{attribute 'linkalways'} 
{attribute 'no_explicit_call' := 'This FB is a CLASS and must be accessed using methods or properties'}
{attribute 'enable_dynamic_creation'}
FUNCTION_BLOCK GetBlueprintsVisitor IMPLEMENTS I_NodeFactoryVisitor, I_NodePrototypeVisitor, I_NodeVisitor, I_ExtensionVisitor, I_InputPortVisitor, I_OutputPortVisitor, I_MetadataVisitor, I_ContentVisitor, I_ParameterVisitor, I_AlarmVisitor
VAR
	serializer : I_Serializer;
END_VAR

METHOD PUBLIC Initialize
VAR_INPUT
	Serializer : I_Serializer;
END_VAR
THIS^.serializer := Serializer;
END_METHOD

METHOD VisitAlarm
VAR_INPUT
	VisitingAlarm : I_Alarm;
END_VAR
serializer.AddString(VisitingAlarm.Message);
END_METHOD

METHOD VisitContent
VAR_INPUT
	VisitingContent : I_Content;
END_VAR
serializer.StartObject();

serializer.AddKeyString('name',VisitingContent.Name);
serializer.Addkey('datatype');
VisitingContent.Data.SerializeTypeWith(serializer);

IF VisitingContent.Metadatum.HasMetadata THEN
	serializer.addkey('metadata');
	serializer.StartArray();
	VisitingContent.Metadatum.Accept(THIS^);
	serializer.EndArray();
END_IF

serializer.EndObject();
END_METHOD

METHOD VisitExtension
VAR_INPUT
	VisitingExtension : I_Extension;
END_VAR
Serializer.StartObject();
Serializer.AddKeyString('name',VisitingExtension.Name);

IF VisitingExtension.Metadatum.HasMetadata THEN
	serializer.addkey('metadata');
	serializer.StartArray();
	VisitingExtension.Metadatum.Accept(THIS^);
	serializer.EndArray();
END_IF

IF VisitingExtension.Alarms.HasAlarms THEN
	serializer.addkey('alarms');
	serializer.StartArray();
	VisitingExtension.Alarms.Accept(THIS^);
	serializer.EndArray();
END_IF

IF VisitingExtension.InputPorts.HasInputPorts THEN
	serializer.addkey('inputPorts');
	serializer.StartArray();
	VisitingExtension.InputPorts.Accept(THIS^);
	serializer.EndArray();
END_IF

IF VisitingExtension.OutputPorts.HasOutputPorts THEN
	serializer.addkey('outputPorts');
	serializer.StartArray();
	VisitingExtension.OutputPorts.Accept(THIS^);
	serializer.EndArray();
END_IF

IF VisitingExtension.Parameters.HasParameters THEN
	serializer.addkey('parameters');
	serializer.StartArray();
	VisitingExtension.Parameters.Accept(THIS^);
	serializer.EndArray();
END_IF

IF VisitingExtension.Contents.HasContents THEN
	serializer.addkey('contents');
	serializer.StartArray();
	VisitingExtension.Parameters.Accept(THIS^);
	serializer.EndArray();
END_IF

Serializer.EndObject();
END_METHOD

METHOD VisitInputPort
VAR_INPUT
	VisitingInputPort : I_InputPort;
END_VAR
serializer.StartObject();

serializer.AddKeyString('name',VisitingInputPort.Name);
serializer.Addkey('datatype');
VisitingInputPort.Data.SerializeTypeWith(serializer);

IF VisitingInputPort.Metadatum.HasMetadata THEN
	serializer.addkey('metadata');
	serializer.StartArray();
	VisitingInputPort.Metadatum.Accept(THIS^);
	serializer.EndArray();
END_IF

serializer.EndObject();
END_METHOD

METHOD VisitMetadatum
VAR_INPUT
	VisitingMetadatum : I_Metadata;
END_VAR
serializer.StartObject();
serializer.AddKeyString('name',VisitingMetadatum.Name);
serializer.AddkeyObject('value',VisitingMetadatum.Data);
serializer.EndObject();
END_METHOD

METHOD VisitNode
VAR_INPUT
	VisitingNode : I_Node;
END_VAR
serializer.StartObject();

IF VisitingNode.Metadatum.HasMetadata THEN
	serializer.addkey('metadata');
	serializer.StartArray();
	VisitingNode.Metadatum.Accept(THIS^);
	serializer.EndArray();
END_IF

IF VisitingNode.Alarms.HasAlarms THEN
	serializer.addkey('alarms');
	serializer.StartArray();
	VisitingNode.Alarms.Accept(THIS^);
	serializer.EndArray();
END_IF

IF VisitingNode.Extensions.HasExtensions THEN
	serializer.addkey('extensions');
	serializer.StartArray();
	VisitingNode.Extensions.Accept(THIS^);
	serializer.EndArray();
END_IF

IF VisitingNode.InputPorts.HasInputPorts THEN
	serializer.addkey('inputPorts');
	serializer.StartArray();
	VisitingNode.InputPorts.Accept(THIS^);
	serializer.EndArray();
END_IF

IF VisitingNode.OutputPorts.HasOutputPorts THEN
	serializer.addkey('outputPorts');
	serializer.StartArray();
	VisitingNode.OutputPorts.Accept(THIS^);
	serializer.EndArray();
END_IF

IF VisitingNode.Parameters.HasParameters THEN
	serializer.addkey('parameters');
	serializer.StartArray();
	VisitingNode.Parameters.Accept(THIS^);
	serializer.EndArray();
END_IF

IF VisitingNode.Contents.HasContents THEN
	serializer.addkey('contents');
	serializer.StartArray();
	VisitingNode.Contents.Accept(THIS^);
	serializer.EndArray();
END_IF

serializer.EndObject();
END_METHOD

METHOD VisitNodeFactory
VAR_INPUT
	VisitingNodeFactory : I_NodeFactory;
END_VAR
serializer.StartObject();
serializer.AddKey('blueprints');
serializer.StartArray();
VisitingNodeFactory.NodePrototypes.Accept(THIS^);
serializer.EndArray();
serializer.EndObject();
END_METHOD

METHOD VisitNodePrototype
VAR_INPUT
	VisitingPrototype : I_NodePrototype;
END_VAR
serializer.StartObject();
serializer.AddKeyString('path',VisitingPrototype.Path);
serializer.AddKey('node');
VisitingPrototype.Node.Accept(THIS^);
serializer.EndObject();
END_METHOD

METHOD VisitOutputPort
VAR_INPUT
	VisitingOutputPort : I_OutputPort;
END_VAR
serializer.StartObject();

serializer.AddKeyString('name',VisitingOutputPort.Name);
serializer.Addkey('datatype');
VisitingOutputPort.Data.SerializeTypeWith(serializer);

IF VisitingOutputPort.Metadatum.HasMetadata THEN
	serializer.addkey('metadata');
	serializer.StartArray();
	VisitingOutputPort.Metadatum.Accept(THIS^);
	serializer.EndArray();
END_IF

serializer.EndObject();
END_METHOD

METHOD VisitParameter
VAR_INPUT
	VisitingProperty : I_Parameter;
END_VAR
serializer.StartObject();

serializer.AddKeyString('name',VisitingProperty.Name);
serializer.Addkey('datatype');
VisitingProperty.Data.SerializeTypeWith(serializer);
serializer.Addkey('defaultValue');
VisitingProperty.Data.SerializeWith(serializer);

IF VisitingProperty.Metadatum.HasMetadata THEN
	serializer.addkey('metadata');
	serializer.StartArray();
	VisitingProperty.Metadatum.Accept(THIS^);
	serializer.EndArray();
END_IF

Serializer.EndObject();
END_METHOD

END_FUNCTION_BLOCK

(* stored: Version 1.1.0.1, ProductVersion 3.1.4024.12
   POU GetBlueprintsVisitor: Id {9a2eaf75-20aa-0bd3-13b7-cac193f2dd25}, SpecialFunc None
   Method Initialize: Id {29462709-d7fd-030c-2f49-7ef200611ec1}
   Method VisitAlarm: Id {9da64f96-4eed-0fb4-1faf-579042990278}
   Method VisitContent: Id {50b7889e-c66a-05bb-2edd-312fd3fc40a8}
   Method VisitExtension: Id {4c5e605f-ae0d-0f06-2bc6-a76c4074af51}
   Method VisitInputPort: Id {04731990-d150-0c09-1976-f0e2a6e832f5}
   Method VisitMetadatum: Id {a5150ceb-d8e0-039b-1117-4915c61d72af}
   Method VisitNode: Id {5dc12cbf-865c-05b7-397f-c3231e60113e}
   Method VisitNodeFactory: Id {2afae386-a62a-0dc0-190f-0b9a578bdd40}
   Method VisitNodePrototype: Id {28145082-70b0-0186-0c74-e7ee1c672bd8}
   Method VisitOutputPort: Id {1e1f3fdb-fb3c-0e29-18d4-eee8d7dddbea}
   Method VisitParameter: Id {8e44ba8a-aa2f-0b5c-3727-b49921055eaf} *)
